PROGRAM P02_GlobalSystemTime
VAR
	fbGlobalTime 		:FB_SystemDateTIme;
END_VAR

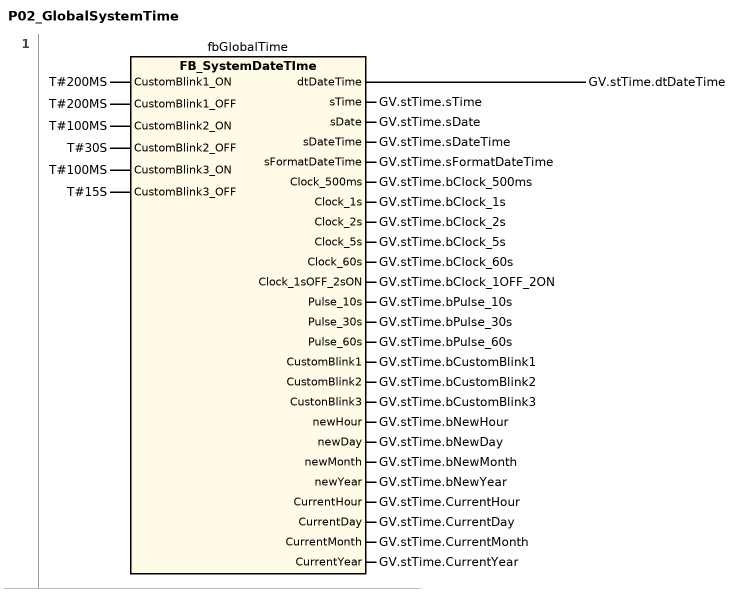
// NETWORK 1
fbGlobalTime(
    CustomBlink1_ON := T#200MS,
    CustomBlink1_OFF := T#200MS,
    CustomBlink2_ON := T#100MS,
    CustomBlink2_OFF := T#30S,
    CustomBlink3_ON := T#100MS,
    CustomBlink3_OFF := T#15S,
    sTime => GV.stTime.sTime,
    sDate => GV.stTime.sDate,
    sDateTime => GV.stTime.sDateTime,
    sFormatDateTime => GV.stTime.sFormatDateTime,
    Clock_500ms => GV.stTime.bClock_500ms,
    Clock_1s => GV.stTime.bClock_1s,
    Clock_2s => GV.stTime.bClock_2s,
    Clock_5s => GV.stTime.bClock_5s,
    Clock_60s => GV.stTime.bClock_60s,
    Clock_1sOFF_2sON => GV.stTime.bClock_1OFF_2ON,
    Pulse_10s => GV.stTime.bPulse_10s,
    Pulse_30s => GV.stTime.bPulse_30s,
    Pulse_60s => GV.stTime.bPulse_60s,
    CustomBlink1 => GV.stTime.bCustomBlink1,
    CustomBlink2 => GV.stTime.bCustomBlink2,
    CustonBlink3 => GV.stTime.bCustomBlink3,
    newHour => GV.stTime.bNewHour,
    newDay => GV.stTime.bNewDay,
    newMonth => GV.stTime.bNewMonth,
    newYear => GV.stTime.bNewYear,
    CurrentHour => GV.stTime.CurrentHour,
    CurrentDay => GV.stTime.CurrentDay,
    CurrentMonth => GV.stTime.CurrentMonth,
    CurrentYear => GV.stTime.CurrentYear); // FB_SystemDateTIme
GV.stTime.dtDateTime := fbGlobalTime.dtDateTime;

END_PROGRAM

(* stored: Version 1.1.0.1
   POU P02_GlobalSystemTime: Id {b84e54e8-046b-4e75-83ca-71c90935ac64}, SpecialFunc None *)
